PROGRAM MAIN
VAR
	StateMachine: FB_StateMachine;
END_VAR

StateMachine(bStart:= Gvl.bStart, bStop:= Gvl.bStop);

GVL.Green := StateMachine.Green;
GVL.Yellow := StateMachine.Yellow;
GVL.Red := StateMachine.Red;

END_PROGRAM

(* stored: Version 1.1.0.1, ProductVersion 3.1.4024.12
   POU MAIN: Id {fc3bf337-a2c5-4f78-93e6-b50f81040e55}, SpecialFunc None *)
